{attribute 'GeneratedUsingTerminal: EL3102--0000'}
{attribute addProperty BoxType "EL3102--0000"}
{attribute addProperty Id "Channel_1AT %I*Channel_7539AA333Channel_2AT %I*Channel_7539AA333WcStateAT %I*WcState_9091E0EB2InfoDataAT %I*InfoData_94A18F5E2"}
{attribute addProperty CRC "1578362931"}
{attribute addProperty Size "10"}
TYPE EL3102_5E13E833 EXTENDS EtcSlaveTerminalBase_947E5A46 :
STRUCT
	{attribute addProperty Name "Channel_1"}
	Channel_1 : Channel_7539AA33;
	{attribute addProperty Name "Channel_2"}
	Channel_2 : Channel_7539AA33;
	{attribute addProperty Name "WcState"}
	WcState : WcState_9091E0EB;
	{attribute addProperty Name "InfoData"}
	InfoData : InfoData_94A18F5E;
END_STRUCT
END_TYPE

(* stored: Version 1.2.0.0, ProductVersion 3.1.4024.9
   DUT EL3102_5E13E833: Id {3da69848-17a6-4a19-b73f-466a6a416659} *)
